(* PLC project Unnamed, Unknown Unnamed 1 *)
(* stored: creationDateTime 2023-04-13T15:52:21, modificationDateTime 2023-04-25T13:16:14 *)

PROGRAM Irrigation_Hardware
  VAR
    OUTLET_VALVE AT %QX0.0 : BOOL;
    OUTLET AT %QX0.1 : BOOL;
    INLET AT %QX0.2 : BOOL;
    INLET_VALVE AT %QX0.3 : BOOL;
    MASTER_COIL AT %QX0.4 : BOOL;
    START AT %IX0.0 : BOOL;
    STOP AT %IX0.1 : BOOL;
    LOW_SENSOR AT %IX0.2 : BOOL;
    HIGH_SENSOR AT %IX0.3 : BOOL;
  END_VAR

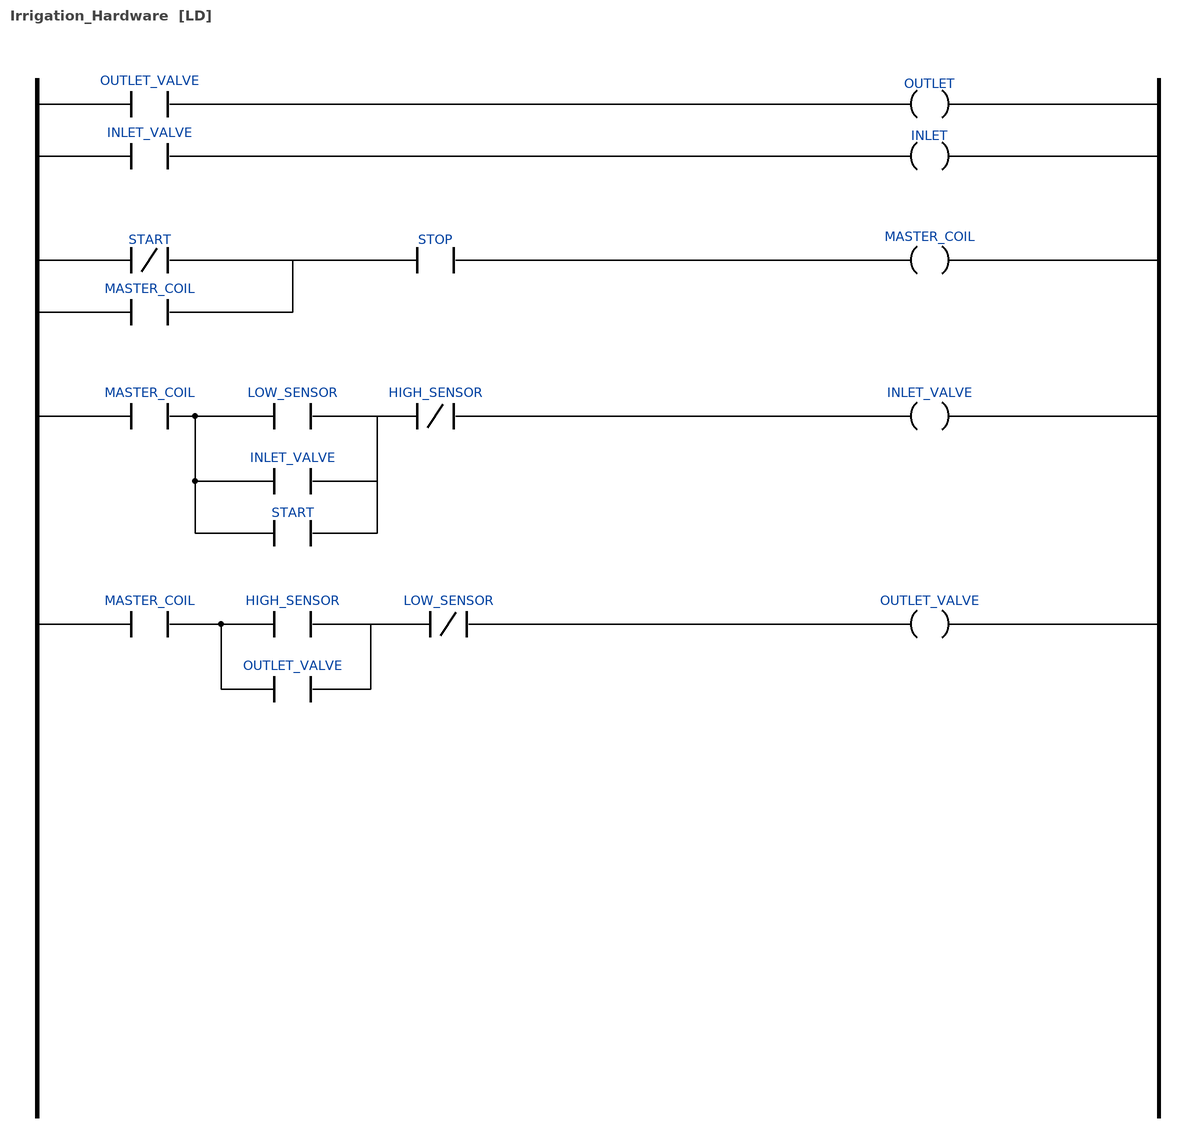
(* LD diagram, written out as Structured Text *)
OUTLET := OUTLET_VALVE;
INLET := INLET_VALVE;
MASTER_COIL := (NOT START OR MASTER_COIL) AND STOP;
INLET_VALVE := MASTER_COIL AND (LOW_SENSOR OR INLET_VALVE OR START) AND NOT HIGH_SENSOR;
OUTLET_VALVE := MASTER_COIL AND (HIGH_SENSOR OR OUTLET_VALVE) AND NOT LOW_SENSOR;
END_PROGRAM

CONFIGURATION Config0
  RESOURCE Res0 ON PLC
    TASK task0(INTERVAL := T#20ms, PRIORITY := 0);
    PROGRAM instance0 WITH task0 : Irrigation_Hardware;
  END_RESOURCE
END_CONFIGURATION
